// Minimal concrete probe for the base classes (Fraktal_QuickStart_and_Suite.md §1).
// Its process logic is only _M_Dispatch. CommandStarts observes the inherited
// command-start callback so the base suite can prove its one-shot semantics.
FUNCTION_BLOCK FB_ProbeCM EXTENDS FB_ControlModuleBase
VAR_INPUT
    SimDone  : BOOL;
    SimFault : BOOL;
    SimState : BOOL;                 // §3.12 the derived fact this probe publishes
    SimPublish : BOOL := TRUE;       // stop publishing to exercise the stale path
END_VAR
VAR_OUTPUT
    CommandStarts : UDINT;
    StateProbe : BOOL;               // what _M_State returned, so the call reads as an assignment
END_VAR

Cyclic();

METHOD Setup : BOOL
VAR_INPUT
    Name : STRING(80);
END_VAR
_M_SetName(Name);
Setup := TRUE;
END_METHOD

METHOD PROTECTED OnCyclic : DINT
OnCyclic := SUPER^.OnCyclic();   // base first (Core §3.14.2)
// §3.12 — a derived flag is published UNCONDITIONALLY every scan. SimPublish exists
// only so the suite can prove what happens when a project breaks that rule.
IF SimPublish THEN
    StateProbe := _M_State(Idx := 1, Key := 'project.test.probeState', Ok := SimState);
END_IF
END_METHOD

METHOD PROTECTED _M_Dispatch
_M_TagCommand(Id := 1, Label := 'PROBE');   // §8.11.4(a) — the one-line command tag
IF SimFault THEN
    _M_Fault(E_Reason.TEST_FAULT, 'probe fault');
ELSIF SimDone THEN
    _M_Complete();
END_IF
END_METHOD

METHOD PROTECTED OnCommandStart : DINT
OnCommandStart := SUPER^.OnCommandStart();
CommandStarts := CommandStarts + 1;
END_METHOD

END_FUNCTION_BLOCK

(* stored: Version 1.1.0.1, ProductVersion 3.1.4024.12
   POU FB_ProbeCM: Id {ace2ffef-da6f-4500-bb16-d6b5e668246d}, SpecialFunc None
   Method Setup: Id {fa777fc7-9e8d-4c24-aab9-7b0fc5bce9d1}
   Method OnCyclic: Id {35959dd2-3c4c-42a7-8c86-2c4db506675f}
   Method _M_Dispatch: Id {09dda4aa-ea32-4a00-b61d-5b786f9f2569}
   Method OnCommandStart: Id {cb7d5d23-6aa4-4636-becb-a6dbc26fb5cb} *)
